PROGRAM MAIN
VAR
	fbTimeDelta : FB_TimeDelta ;
	bStartButton : BOOL;
	bStopButton : BOOL;
	DisplayDeltaTime : ST_TimeStruct;
	bStartButtonPressed : BOOL := FALSE; // Latch for Start button
    bStopButtonPressed : BOOL := FALSE;  // Latch for Stop button
	bReset : BOOL;
END_VAR

fbTimeDelta();

// Logic for Start Button
IF bStartButton AND NOT bStartButtonPressed THEN
    fbTimeDelta.Start(); // Record the start time
    bStartButtonPressed := TRUE; // Latch the start button
END_IF

// Reset the latch if the button is released
IF NOT bStartButton THEN
    bStartButtonPressed := FALSE;
END_IF

// Logic for Stop Button
IF bStopButton AND NOT bStopButtonPressed THEN
    fbTimeDelta.Stop(); // Record the stop time
    bStopButtonPressed := TRUE; // Latch the stop button
    
    // Calculate and display the delta time
    DisplayDeltaTime := fbTimeDelta.GetDelta();
END_IF

// Reset the latch if the button is released
IF NOT bStopButton THEN
    bStopButtonPressed := FALSE;
END_IF

END_PROGRAM

(* stored: Version 1.1.0.1, ProductVersion 3.1.4024.12
   POU MAIN: Id {78d2917f-3efd-400c-b9b5-d7f9be5bc87b}, SpecialFunc None *)
